INTERFACE I_Enumerable EXTENDS I_Object

METHOD ForEach : I_Enumerable
VAR_INPUT
    ipAction: I_Action;
END_VAR
END_METHOD

END_INTERFACE

(* stored: Version 1.1.0.1, ProductVersion 3.1.4024.12
   Itf I_Enumerable: Id {77cfedcd-ab49-4197-ba6c-31599fc7655f}
   Method ForEach: Id {3d77c5da-1a0e-4f98-a6d1-ea12d80627a3} *)
